FUNCTION_BLOCK FB_BasicAxisFFO
(*
    Placeholder FFO logic for no beam allowed, pre-comissioning

    Fast fault is applied if the axis is moving.
*)
VAR_IN_OUT
    Axis: AXIS_REF;
    fbFFHWO: FB_HardwareFFOutput;
END_VAR
VAR_INPUT
    sName: STRING;
END_VAR
VAR_OUTPUT
    bIsNotMoving: BOOL;
END_VAR
VAR
    fbFF: FB_FastFault := (i_Desc := 'Device is moving',
                           i_TypeCode := 16#2100,
                           i_xAutoReset := TRUE);
END_VAR

bIsNotMoving := NOT Axis.Status.Moving;
fbFF(i_DevName := sName,
     i_xOK := bIsNotMoving,
     io_fbFFHWO := fbFFHWO);

END_FUNCTION_BLOCK

(* stored: Version 1.1.0.1, ProductVersion 3.1.4022.18
   POU FB_BasicAxisFFO: Id {43d7d8ae-9dd2-073d-2b53-53a6782f7ace}, SpecialFunc None *)
